// Mitsubishi GX Works2 project: 0630실린더 응용동작3 3초 대기   PLC: Q02/Q02H

PROGRAM MAIN
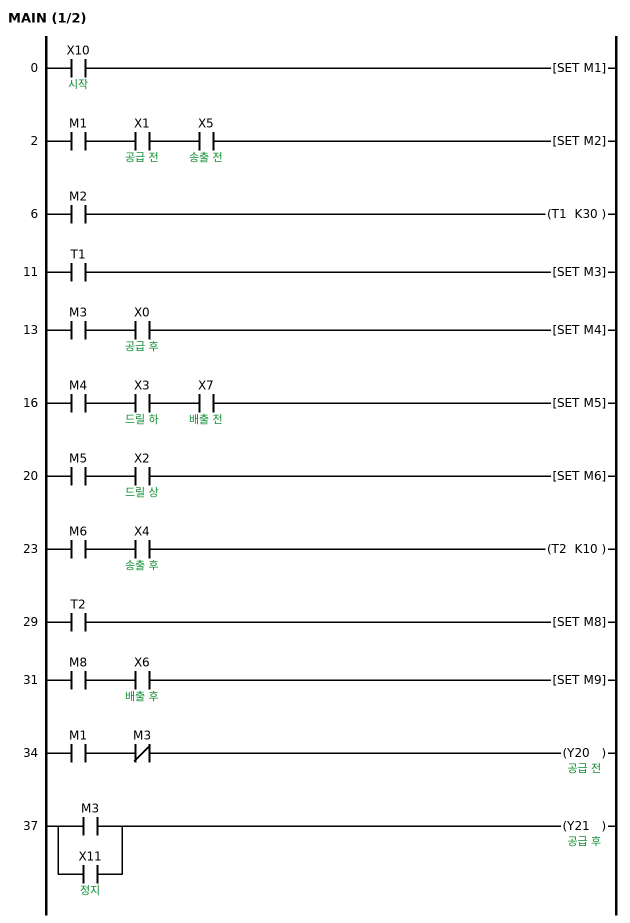
0     LD      X10  ; 시작
      SET     M1
2     LD      M1
      AND     X1  ; 공급 전
      AND     X5  ; 송출 전
      SET     M2
6     LD      M2
      OUT     T1 K30
11    LD      T1
      SET     M3
13    LD      M3
      AND     X0  ; 공급 후
      SET     M4
16    LD      M4
      AND     X3  ; 드릴 하
      AND     X7  ; 배출 전
      SET     M5
20    LD      M5
      AND     X2  ; 드릴 상
      SET     M6
23    LD      M6
      AND     X4  ; 송출 후
      OUT     T2 K10
29    LD      T2
      SET     M8
31    LD      M8
      AND     X6  ; 배출 후
      SET     M9
34    LD      M1
      ANI     M3
      OUT     Y20  ; 공급 전
37    LD      M3
      OR      X11  ; 정지
      OUT     Y21  ; 공급 후
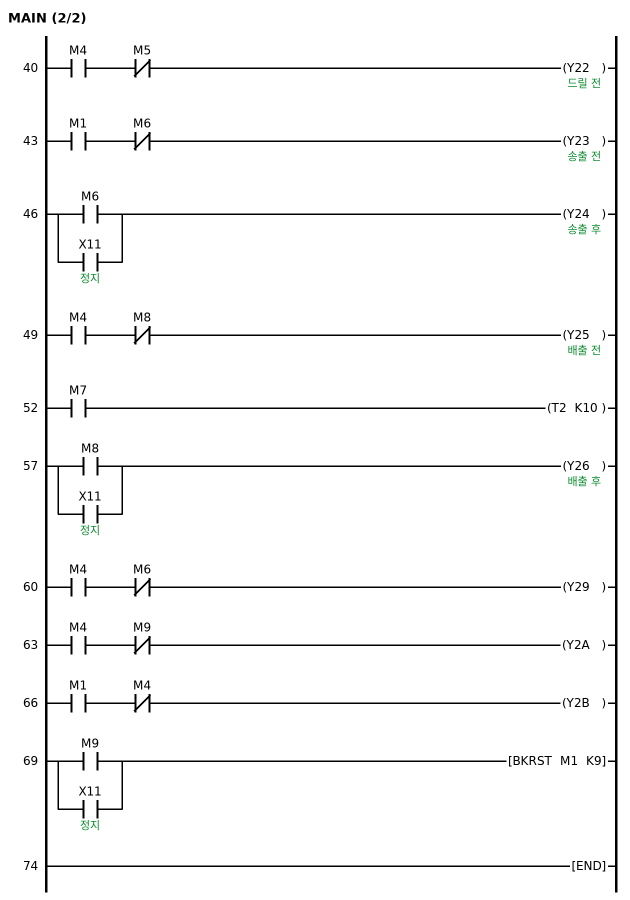
40    LD      M4
      ANI     M5
      OUT     Y22  ; 드릴 전
43    LD      M1
      ANI     M6
      OUT     Y23  ; 송출 전
46    LD      M6
      OR      X11  ; 정지
      OUT     Y24  ; 송출 후
49    LD      M4
      ANI     M8
      OUT     Y25  ; 배출 전
52    LD      M7
      OUT     T2 K10
57    LD      M8
      OR      X11  ; 정지
      OUT     Y26  ; 배출 후
60    LD      M4
      ANI     M6
      OUT     Y29
63    LD      M4
      ANI     M9
      OUT     Y2A
66    LD      M1
      ANI     M4
      OUT     Y2B
69    LD      M9
      OR      X11  ; 정지
      BKRST   M1 K9
74    END
END_PROGRAM
